(* PLC project Untitled1, Beckhoff Automation GmbH TF6420 Database Server Query Analyser 1.0.0.0 *)
(* stored: creationDateTime 2016-05-17T16:57:53, modificationDateTime 2016-05-17T16:57:53 *)

TYPE ST_DB_Enthalpie_r134a : STRUCT
  id : DINT;
  timestamp : DT;
  Temperatur : STRING(45);
  h1 : STRING(45);
  h2 : STRING(45);
  h3 : STRING(45);
  h4 : STRING(45);
  h5 : STRING(45);
  h6 : STRING(45);
  h7 : STRING(45);
  h8 : STRING(45);
  h9 : STRING(45);
  h10 : STRING(45);
  h11 : STRING(45);
  h12 : STRING(45);
  h13 : STRING(45);
  h14 : STRING(45);
  h15 : STRING(45);
END_STRUCT;
END_TYPE
